TYPE ST_MESSAGE_INFO :
STRUCT
	tTimestamp 	 : DT;
	sDescription : T_MaxString;
	eOperation 	 : E_OPERATION;
END_STRUCT
END_TYPE

(* stored: Version 1.1.0.1, ProductVersion 3.1.4024.12
   DUT ST_MESSAGE_INFO: Id {993d31d7-12ab-423f-83b3-d2bab03868cd} *)
